// TIA Portal V20 export
FUNCTION "CallCounterMapping" : Void   // FC94, LAD
// stored: SetENOAutomatically false
   VAR CONSTANT
      TRUE : Bool := TRUE;
   END_VAR
BEGIN

REGION Network 1: Input Qty
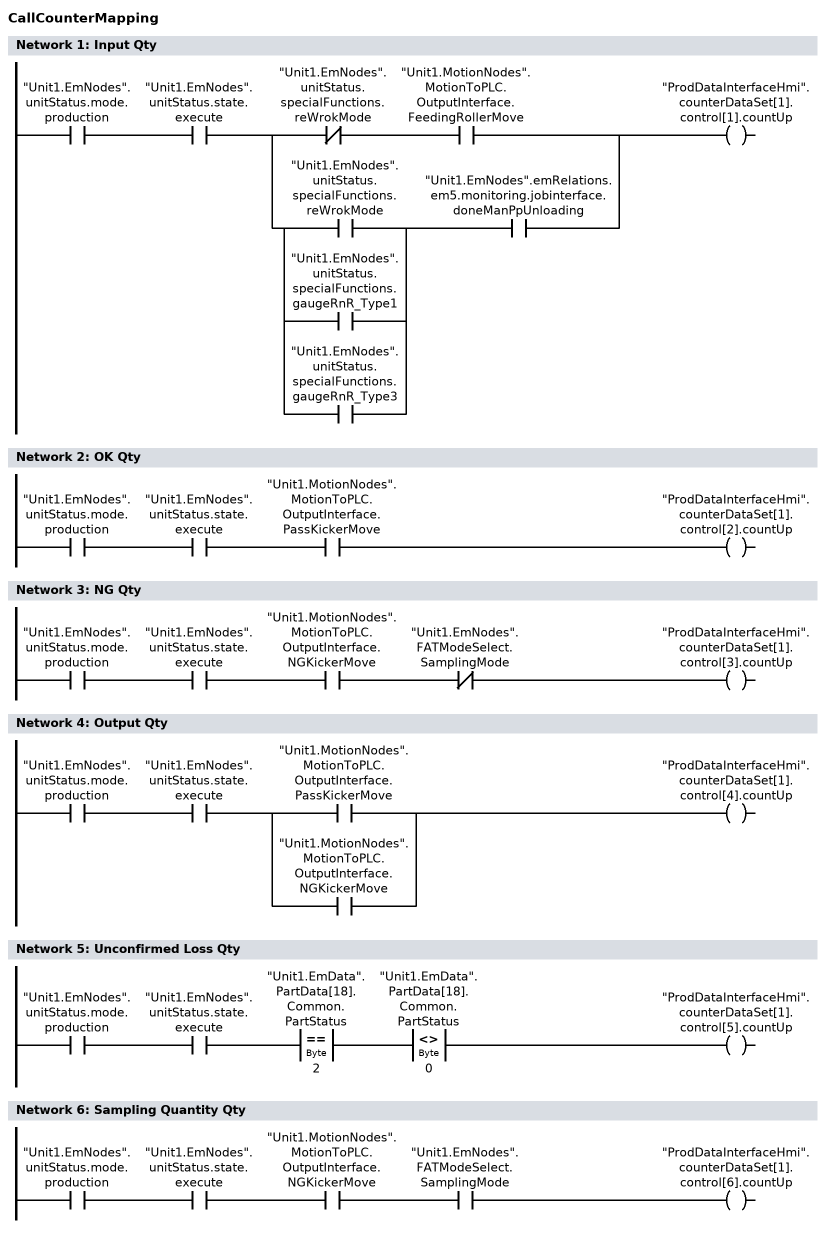
   RUNG wire#powerrail
      Contact( "Unit1.EmNodes".unitStatus.mode.production )
      Contact( "Unit1.EmNodes".unitStatus.state.execute )
      wire#w1
      I_Contact( "Unit1.EmNodes".unitStatus.specialFunctions.reWrokMode )
      Contact( "Unit1.MotionNodes".MotionToPLC.OutputInterface.FeedingRollerMove )
      wire#w2
      Coil( "ProdDataInterfaceHmi".counterDataSet[1].control[1].countUp )
   END_RUNG
   RUNG wire#w1
      Contact( "Unit1.EmNodes".unitStatus.specialFunctions.reWrokMode )
      wire#w3
      Contact( "Unit1.EmNodes".emRelations.em5.monitoring.jobinterface.doneManPpUnloading )
   END_RUNG wire#w2
   RUNG wire#w1
      Contact( "Unit1.EmNodes".unitStatus.specialFunctions.gaugeRnR_Type1 )
   END_RUNG wire#w3
   RUNG wire#w1
      Contact( "Unit1.EmNodes".unitStatus.specialFunctions.gaugeRnR_Type3 )
   END_RUNG wire#w3
   // the same network as SCL:
   "ProdDataInterfaceHmi".counterDataSet[1].control[1].countUp := "Unit1.EmNodes".unitStatus.mode.production AND "Unit1.EmNodes".unitStatus.state.execute AND ((NOT "Unit1.EmNodes".unitStatus.specialFunctions.reWrokMode AND "Unit1.MotionNodes".MotionToPLC.OutputInterface.FeedingRollerMove) OR (("Unit1.EmNodes".unitStatus.specialFunctions.reWrokMode OR "Unit1.EmNodes".unitStatus.specialFunctions.gaugeRnR_Type1 OR "Unit1.EmNodes".unitStatus.specialFunctions.gaugeRnR_Type3) AND "Unit1.EmNodes".emRelations.em5.monitoring.jobinterface.doneManPpUnloading));
END_REGION

REGION Network 2: OK Qty
   RUNG wire#powerrail
      Contact( "Unit1.EmNodes".unitStatus.mode.production )
      Contact( "Unit1.EmNodes".unitStatus.state.execute )
      Contact( "Unit1.MotionNodes".MotionToPLC.OutputInterface.PassKickerMove )
      Coil( "ProdDataInterfaceHmi".counterDataSet[1].control[2].countUp )
   END_RUNG
   // the same network as SCL:
   "ProdDataInterfaceHmi".counterDataSet[1].control[2].countUp := "Unit1.EmNodes".unitStatus.mode.production AND "Unit1.EmNodes".unitStatus.state.execute AND "Unit1.MotionNodes".MotionToPLC.OutputInterface.PassKickerMove;
END_REGION

REGION Network 3: NG Qty
   RUNG wire#powerrail
      Contact( "Unit1.EmNodes".unitStatus.mode.production )
      Contact( "Unit1.EmNodes".unitStatus.state.execute )
      Contact( "Unit1.MotionNodes".MotionToPLC.OutputInterface.NGKickerMove )
      I_Contact( "Unit1.EmNodes".FATModeSelect.SamplingMode )
      Coil( "ProdDataInterfaceHmi".counterDataSet[1].control[3].countUp )
   END_RUNG
   // the same network as SCL:
   "ProdDataInterfaceHmi".counterDataSet[1].control[3].countUp := "Unit1.EmNodes".unitStatus.mode.production AND "Unit1.EmNodes".unitStatus.state.execute AND "Unit1.MotionNodes".MotionToPLC.OutputInterface.NGKickerMove AND NOT "Unit1.EmNodes".FATModeSelect.SamplingMode;
END_REGION

REGION Network 4: Output Qty
   RUNG wire#powerrail
      Contact( "Unit1.EmNodes".unitStatus.mode.production )
      Contact( "Unit1.EmNodes".unitStatus.state.execute )
      wire#w1
      Contact( "Unit1.MotionNodes".MotionToPLC.OutputInterface.PassKickerMove )
      wire#w2
      Coil( "ProdDataInterfaceHmi".counterDataSet[1].control[4].countUp )
   END_RUNG
   RUNG wire#w1
      Contact( "Unit1.MotionNodes".MotionToPLC.OutputInterface.NGKickerMove )
   END_RUNG wire#w2
   // the same network as SCL:
   "ProdDataInterfaceHmi".counterDataSet[1].control[4].countUp := "Unit1.EmNodes".unitStatus.mode.production AND "Unit1.EmNodes".unitStatus.state.execute AND ("Unit1.MotionNodes".MotionToPLC.OutputInterface.PassKickerMove OR "Unit1.MotionNodes".MotionToPLC.OutputInterface.NGKickerMove);
END_REGION

REGION Network 5: Unconfirmed Loss Qty
   RUNG wire#powerrail
      Contact( "Unit1.EmNodes".unitStatus.mode.production )
      Contact( "Unit1.EmNodes".unitStatus.state.execute )
      { S7_Templates := "SrcType := Byte" } EQ_Contact(in1 := "Unit1.EmData".PartData[18].Common.PartStatus, in2 := 2)
      { S7_Templates := "SrcType := Byte" } NE_Contact(in1 := "Unit1.EmData".PartData[18].Common.PartStatus, in2 := 0)
      Coil( "ProdDataInterfaceHmi".counterDataSet[1].control[5].countUp )
   END_RUNG
   // the same network as SCL:
   "ProdDataInterfaceHmi".counterDataSet[1].control[5].countUp := "Unit1.EmNodes".unitStatus.mode.production AND "Unit1.EmNodes".unitStatus.state.execute AND ("Unit1.EmData".PartData[18].Common.PartStatus = 2) AND ("Unit1.EmData".PartData[18].Common.PartStatus <> 0);
END_REGION

REGION Network 6: Sampling Quantity Qty
   RUNG wire#powerrail
      Contact( "Unit1.EmNodes".unitStatus.mode.production )
      Contact( "Unit1.EmNodes".unitStatus.state.execute )
      Contact( "Unit1.MotionNodes".MotionToPLC.OutputInterface.NGKickerMove )
      Contact( "Unit1.EmNodes".FATModeSelect.SamplingMode )
      Coil( "ProdDataInterfaceHmi".counterDataSet[1].control[6].countUp )
   END_RUNG
   // the same network as SCL:
   "ProdDataInterfaceHmi".counterDataSet[1].control[6].countUp := "Unit1.EmNodes".unitStatus.mode.production AND "Unit1.EmNodes".unitStatus.state.execute AND "Unit1.MotionNodes".MotionToPLC.OutputInterface.NGKickerMove AND "Unit1.EmNodes".FATModeSelect.SamplingMode;
END_REGION
END_FUNCTION
